FUNCTION_BLOCK CU010ManualTask EXTENDS TcoTaskedService IMPLEMENTS ICUTask
VAR
END_VAR

Run();

(*~
	<docu>
		<summary>
			Main method of the sequener. Custom code needs to be placed here. The sequencer is executed by call of **Instance.Run()** method.
			This method is abstract, and it must be overridden in derived block.
		</summary>
	</docu>
~*)
METHOD PROTECTED Main : BOOL
Messenger.Notify('Running manual mode');
Station.Components.Group1.horizontalCylinder.Service();
END_METHOD

METHOD PROTECTED OnStart
Station.AutomatTask.Restore();
Station.GroundTask.Restore();
Station.GroundTask.CancelGround();
END_METHOD

PROPERTY Station : REFERENCE TO CU010
GET
VAR
    _station : POINTER TO CU010;
END_VAR
IF __QUERYPOINTER(Parent, _station) THEN // Check if _Parent is Station001
    Station REF= _station^;              // If the check is successful dereference a pointer. simlar to THIS^ or SUPER^
END_IF
END_GET
END_PROPERTY

END_FUNCTION_BLOCK

(* stored: Version 1.1.0.1
   POU CU010ManualTask: Id {3067a6bb-2116-489c-8f77-ec88d28bd912}, SpecialFunc None
   Method Main: Id {86c0a293-e0bf-4742-96d4-6a5351013ec0}
   Method OnStart: Id {4400aae1-6660-4bbe-85c5-ef5993a0ea80}
   Property Station: Id {3daf9692-5397-45f9-a23f-6c342bf12bd1}
   Get Get: Id {c786ace9-bf2b-4715-8cb3-9256add4c5e0} *)
